Fanuc KAREL source: kb00158.KL

-- PROVISIONAL review KL for V1013-1; original PC SHA256 341912840e6903eeb8cc54235271077eea366581f0db57cc32eb1f88ca070542
-- Incomplete behavior may be omitted. Consult companion uncertainty JSON. Do not deploy.
PROGRAM KB00158
%NOLOCKGROUP
BEGIN
  -- UNRESOLVED_PC offsets 5-12; opcodes 9D,23
  -- UNRESOLVED_PC offsets 17-24; opcodes 9D,23
  -- UNRESOLVED_PC offsets 29-45; opcodes 27,22,22,31
  -- UNRESOLVED_PC offsets 50-54; opcodes 7F
END KB00158
